FUNCTION_BLOCK TcoDigitalInspector EXTENDS TcoCore.TcoObject

METHOD Inspect : BOOL
VAR_INPUT
	inValue : BOOL;
END_VAR
END_METHOD

END_FUNCTION_BLOCK

(* stored: Version 1.1.0.1, ProductVersion 3.1.4024.9
   POU TcoDigitalInspector: Id {b1413ab6-cf32-03b8-31af-46a8ec8720ab}, SpecialFunc None
   Method Inspect: Id {304a74e1-ec39-09fd-0ecf-8a74644a243b} *)
